// TIA Portal V21 export
FUNCTION_BLOCK "SIP TEMPERATURE CONTROLER"   // FB502, LAD
{ S7_Optimized_Access := 'FALSE' }
// stored: AutoNumber false, SetENOAutomatically false
   VAR_INPUT
      "CONROL ON" : Bool;
      Second_Pulse : Bool;
      Actual_sip_temp : Real;
      "SET  TEMPERATUR" : Real;
      "TEMPERATURE RANGE_1" : Real;
      "TEMPERATURE RANGE_2" : Real;
      "TEMPERATURE RANGE_4" : Real;
      "TEMPERATURE RANGE_6" : Real;
      "TEMPERATURE RANGE_8" : Real;
      ON_SEC_1 { ExternalAccessible := 'False'; ExternalVisible := 'False'; ExternalWritable := 'False'} : Int;
      ON_SEC_2 { ExternalAccessible := 'False'; ExternalVisible := 'False'; ExternalWritable := 'False'} : Int;
      ON_SEC_3 { ExternalAccessible := 'False'; ExternalVisible := 'False'; ExternalWritable := 'False'} : Int;
      ON_SEC_4 { ExternalAccessible := 'False'; ExternalVisible := 'False'; ExternalWritable := 'False'} : Int;
      OFF_SEC_1 { ExternalAccessible := 'False'; ExternalVisible := 'False'; ExternalWritable := 'False'} : Int;
      OFF_SEC_2 { ExternalAccessible := 'False'; ExternalVisible := 'False'; ExternalWritable := 'False'} : Int;
      OFF_SEC_3 { ExternalAccessible := 'False'; ExternalVisible := 'False'; ExternalWritable := 'False'} : Int;
      OFF_SEC_4 { ExternalAccessible := 'False'; ExternalVisible := 'False'; ExternalWritable := 'False'} : Int;
      RESET_BIT : Bool;
   END_VAR
   VAR_OUTPUT
      "VALVE CONTROL" : Bool;
      TEMPPERATUR_REACHED : Bool;
   END_VAR
   VAR_IN_OUT
      ON_SEC : Int;
      OFF_SEC : Int;
      ON_SEC_TIME : Int;
      OFF_SEC_TIME : Int;
      TEMP_1 : Bool;
   END_VAR
   VAR_TEMP   // added for the SCL form of the ladder/FBD networks
      _w1 : Bool;
      _w2 : Bool;
      _w3 : Bool;
   END_VAR
BEGIN

REGION Network 1: range
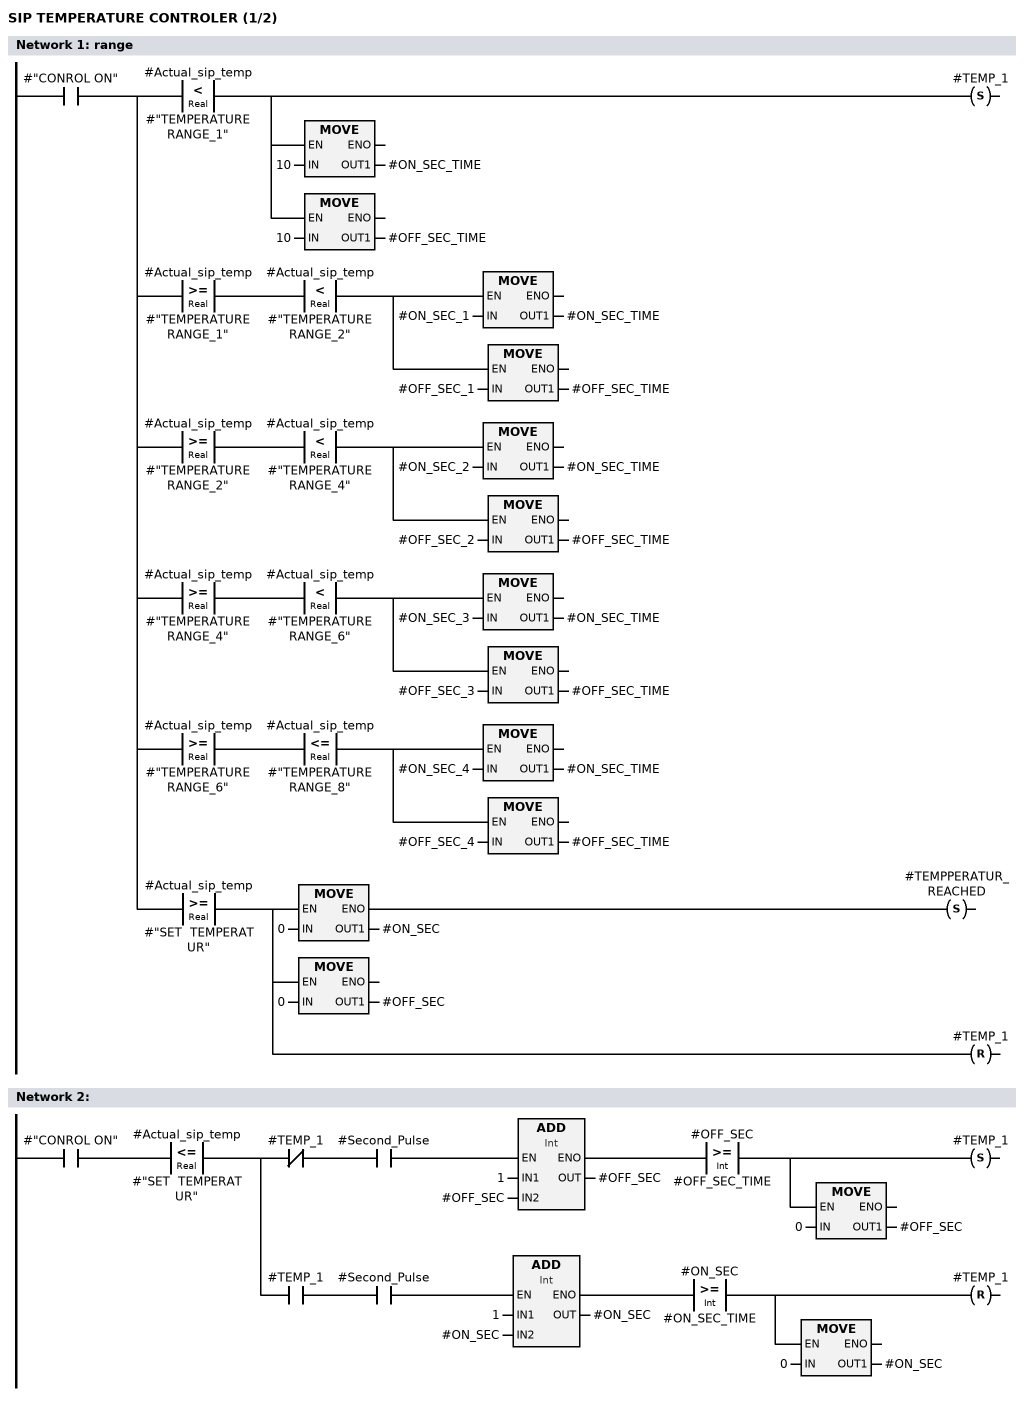
   RUNG wire#powerrail
      Contact( #"CONROL ON" )
      wire#w1
      { S7_Templates := "SrcType := Real" } LT_Contact(in1 := #Actual_sip_temp, in2 := #"TEMPERATURE RANGE_1")
      wire#w2
      S_Coil( #TEMP_1 )
   END_RUNG
   RUNG wire#w2
      { S7_GenerateENO := "TRUE" } Move(in := 10, out1 => #ON_SEC_TIME)
   END_RUNG
   RUNG wire#w2
      { S7_GenerateENO := "TRUE" } Move(in := 10, out1 => #OFF_SEC_TIME)
   END_RUNG
   RUNG wire#w1
      { S7_Templates := "SrcType := Real" } GE_Contact(in1 := #Actual_sip_temp, in2 := #"TEMPERATURE RANGE_1")
      { S7_Templates := "SrcType := Real" } LT_Contact(in1 := #Actual_sip_temp, in2 := #"TEMPERATURE RANGE_2")
      wire#w3
      { S7_GenerateENO := "TRUE" } Move(in := #ON_SEC_1, out1 => #ON_SEC_TIME)
   END_RUNG
   RUNG wire#w3
      { S7_GenerateENO := "TRUE" } Move(in := #OFF_SEC_1, out1 => #OFF_SEC_TIME)
   END_RUNG
   RUNG wire#w1
      { S7_Templates := "SrcType := Real" } GE_Contact(in1 := #Actual_sip_temp, in2 := #"TEMPERATURE RANGE_2")
      { S7_Templates := "SrcType := Real" } LT_Contact(in1 := #Actual_sip_temp, in2 := #"TEMPERATURE RANGE_4")
      wire#w4
      { S7_GenerateENO := "TRUE" } Move(in := #ON_SEC_2, out1 => #ON_SEC_TIME)
   END_RUNG
   RUNG wire#w4
      { S7_GenerateENO := "TRUE" } Move(in := #OFF_SEC_2, out1 => #OFF_SEC_TIME)
   END_RUNG
   RUNG wire#w1
      { S7_Templates := "SrcType := Real" } GE_Contact(in1 := #Actual_sip_temp, in2 := #"TEMPERATURE RANGE_4")
      { S7_Templates := "SrcType := Real" } LT_Contact(in1 := #Actual_sip_temp, in2 := #"TEMPERATURE RANGE_6")
      wire#w5
      { S7_GenerateENO := "TRUE" } Move(in := #ON_SEC_3, out1 => #ON_SEC_TIME)
   END_RUNG
   RUNG wire#w5
      { S7_GenerateENO := "TRUE" } Move(in := #OFF_SEC_3, out1 => #OFF_SEC_TIME)
   END_RUNG
   RUNG wire#w1
      { S7_Templates := "SrcType := Real" } GE_Contact(in1 := #Actual_sip_temp, in2 := #"TEMPERATURE RANGE_6")
      { S7_Templates := "SrcType := Real" } LE_Contact(in1 := #Actual_sip_temp, in2 := #"TEMPERATURE RANGE_8")
      wire#w6
      { S7_GenerateENO := "TRUE" } Move(in := #ON_SEC_4, out1 => #ON_SEC_TIME)
   END_RUNG
   RUNG wire#w6
      { S7_GenerateENO := "TRUE" } Move(in := #OFF_SEC_4, out1 => #OFF_SEC_TIME)
   END_RUNG
   RUNG wire#w1
      { S7_Templates := "SrcType := Real" } GE_Contact(in1 := #Actual_sip_temp, in2 := #"SET  TEMPERATUR")
      wire#w7
      { S7_GenerateENO := "TRUE" } Move(in := 0, out1 => #ON_SEC)
      S_Coil( #TEMPPERATUR_REACHED )
   END_RUNG
   RUNG wire#w7
      { S7_GenerateENO := "TRUE" } Move(in := 0, out1 => #OFF_SEC)
   END_RUNG
   RUNG wire#w7
      R_Coil( #TEMP_1 )
   END_RUNG
   // the same network as SCL:
   // ENO of a box is taken as its EN; it also drops when the box reports an error
   IF #"CONROL ON" AND (#Actual_sip_temp < #"TEMPERATURE RANGE_1") THEN
       #TEMP_1 := TRUE;
       #ON_SEC_TIME := 10;
       #OFF_SEC_TIME := 10;
   END_IF;
   IF #"CONROL ON" AND (#Actual_sip_temp >= #"TEMPERATURE RANGE_1") AND (#Actual_sip_temp < #"TEMPERATURE RANGE_2") THEN
       #ON_SEC_TIME := #ON_SEC_1;
       #OFF_SEC_TIME := #OFF_SEC_1;
   END_IF;
   IF #"CONROL ON" AND (#Actual_sip_temp >= #"TEMPERATURE RANGE_2") AND (#Actual_sip_temp < #"TEMPERATURE RANGE_4") THEN
       #ON_SEC_TIME := #ON_SEC_2;
       #OFF_SEC_TIME := #OFF_SEC_2;
   END_IF;
   IF #"CONROL ON" AND (#Actual_sip_temp >= #"TEMPERATURE RANGE_4") AND (#Actual_sip_temp < #"TEMPERATURE RANGE_6") THEN
       #ON_SEC_TIME := #ON_SEC_3;
       #OFF_SEC_TIME := #OFF_SEC_3;
   END_IF;
   IF #"CONROL ON" AND (#Actual_sip_temp >= #"TEMPERATURE RANGE_6") AND (#Actual_sip_temp <= #"TEMPERATURE RANGE_8") THEN
       #ON_SEC_TIME := #ON_SEC_4;
       #OFF_SEC_TIME := #OFF_SEC_4;
   END_IF;
   IF #"CONROL ON" AND (#Actual_sip_temp >= #"SET  TEMPERATUR") THEN
       #ON_SEC := 0;
       #TEMPPERATUR_REACHED := TRUE;
       #OFF_SEC := 0;
       #TEMP_1 := FALSE;
   END_IF;
END_REGION

REGION Network 2
   RUNG wire#powerrail
      Contact( #"CONROL ON" )
      { S7_Templates := "SrcType := Real" } LE_Contact(in1 := #Actual_sip_temp, in2 := #"SET  TEMPERATUR")
      wire#w1
      I_Contact( #TEMP_1 )
      Contact( #Second_Pulse )
      { S7_Templates := "SrcType := Int"; S7_GenerateENO := "TRUE" } Add(in1 := 1, in2 := #OFF_SEC, out => #OFF_SEC)
      { S7_Templates := "SrcType := Int" } GE_Contact(in1 := #OFF_SEC, in2 := #OFF_SEC_TIME)
      wire#w2
      S_Coil( #TEMP_1 )
   END_RUNG
   RUNG wire#w2
      { S7_GenerateENO := "TRUE" } Move(in := 0, out1 => #OFF_SEC)
   END_RUNG
   RUNG wire#w1
      Contact( #TEMP_1 )
      Contact( #Second_Pulse )
      { S7_Templates := "SrcType := Int"; S7_GenerateENO := "TRUE" } Add(in1 := 1, in2 := #ON_SEC, out => #ON_SEC)
      { S7_Templates := "SrcType := Int" } GE_Contact(in1 := #ON_SEC, in2 := #ON_SEC_TIME)
      wire#w3
      R_Coil( #TEMP_1 )
   END_RUNG
   RUNG wire#w3
      { S7_GenerateENO := "TRUE" } Move(in := 0, out1 => #ON_SEC)
   END_RUNG
   // the same network as SCL:
   // ENO of a box is taken as its EN; it also drops when the box reports an error
   #_w1 := #"CONROL ON" AND (#Actual_sip_temp <= #"SET  TEMPERATUR");
   #_w2 := #_w1 AND NOT #TEMP_1 AND #Second_Pulse;
   IF #_w2 THEN #OFF_SEC := 1 + #OFF_SEC; END_IF;
   IF #_w2 AND (#OFF_SEC >= #OFF_SEC_TIME) THEN
       #TEMP_1 := TRUE;
       #OFF_SEC := 0;
   END_IF;
   #_w3 := #_w1 AND #TEMP_1 AND #Second_Pulse;
   IF #_w3 THEN #ON_SEC := 1 + #ON_SEC; END_IF;
   IF #_w3 AND (#ON_SEC >= #ON_SEC_TIME) THEN
       #TEMP_1 := FALSE;
       #ON_SEC := 0;
   END_IF;
END_REGION

REGION Network 3
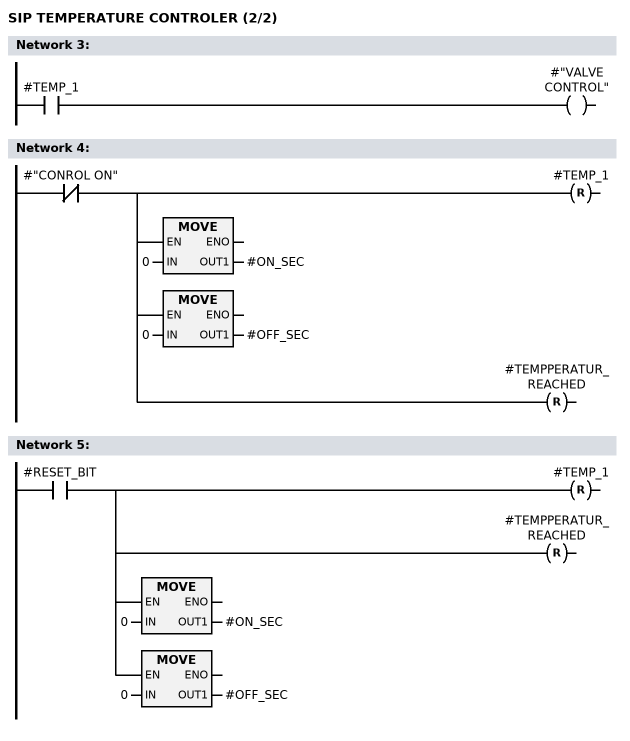
   RUNG wire#powerrail
      Contact( #TEMP_1 )
      Coil( #"VALVE CONTROL" )
   END_RUNG
   // the same network as SCL:
   #"VALVE CONTROL" := #TEMP_1;
END_REGION

REGION Network 4
   RUNG wire#powerrail
      I_Contact( #"CONROL ON" )
      wire#w1
      R_Coil( #TEMP_1 )
   END_RUNG
   RUNG wire#w1
      { S7_GenerateENO := "TRUE" } Move(in := 0, out1 => #ON_SEC)
   END_RUNG
   RUNG wire#w1
      { S7_GenerateENO := "TRUE" } Move(in := 0, out1 => #OFF_SEC)
   END_RUNG
   RUNG wire#w1
      R_Coil( #TEMPPERATUR_REACHED )
   END_RUNG
   // the same network as SCL:
   IF NOT #"CONROL ON" THEN
       #TEMP_1 := FALSE;
       #ON_SEC := 0;
       #OFF_SEC := 0;
       #TEMPPERATUR_REACHED := FALSE;
   END_IF;
END_REGION

REGION Network 5
   RUNG wire#powerrail
      Contact( #RESET_BIT )
      wire#w1
      R_Coil( #TEMP_1 )
   END_RUNG
   RUNG wire#w1
      R_Coil( #TEMPPERATUR_REACHED )
   END_RUNG
   RUNG wire#w1
      { S7_GenerateENO := "TRUE" } Move(in := 0, out1 => #ON_SEC)
   END_RUNG
   RUNG wire#w1
      { S7_GenerateENO := "TRUE" } Move(in := 0, out1 => #OFF_SEC)
   END_RUNG
   // the same network as SCL:
   IF #RESET_BIT THEN
       #TEMP_1 := FALSE;
       #TEMPPERATUR_REACHED := FALSE;
       #ON_SEC := 0;
       #OFF_SEC := 0;
   END_IF;
END_REGION
END_FUNCTION_BLOCK
